Staubli VAL3: loadNext.pgx

program loadNext(string x_sPage, string& x_sItems[])
// load the next page
  local num i
  local string l_sMessage
begin
  // look if the page libload is correct
  i=page:libLoad(x_sPage)
  delay(0)
  if i!=0
    logMsg("[KERNEL] INTERFACE:PAGE LIBLOAD "+x_sPage+" result "+toString("",i))
    call language:message(l_sMessage,-7)
    popUpMsg(l_sMessage+x_sPage+" ; "+toString("",i))
  else
    // copy all the field from x_sItems to the next page
    call use:stringCopy(x_sItems,page:sItems)
    call page:main()
  endIf
end
